Universal Robots PolyScope program: g_2.urp

Program g_2 (installation=string_planes directory=/programs createdIn=5.17.3 lastSavedIn=5.17.3 robotSerialNumber=20245501435)
Calibrated DH parameters: a=[0.000154, -0.137004, -0.385524, -0.00002, 0.000092, 0]; d=[0.162441, 211.794786, -230.585024, 18.923638, 0.099786, 0.09951]; alpha=[1.569493, -0.001902, 0.003874, 1.570111, -1.570167, 0]; deltaTheta=[0, -1.242934, 1.056292, 0.186646, 0.000002, 0.000001]
InitVariablesNode
Robot Program (runOnlyOnce=false)
  MoveL speed 250 mm/s, acceleration 1200 mm/s^2 (useActiveTCP=true) feature=Plane_3
    Waypoint Waypoint_1: TCP in base x=347.51 y=672.22 z=96.15 mm, rx=-1.6525 ry=-1.6511 rz=0.6428 rad; joints [-132.145, -24.912, 67.944, -99.663, -48.733, -144.753] deg; TCP offset x=28.21 y=-96.107 z=-99.69 mm, rx=0 ry=0 rz=0 rad; feature pose in base x=319.452 y=675.799 z=94.591 mm, rx=2.7302 ry=-0.0495 rz=1.4252 rad
    Waypoint Waypoint_2 (Relative): relativeFromPosition TCP in base x=347.532 y=672.21 z=96.159 mm, rx=-1.6525 ry=-1.6511 rz=0.6428 rad; joints [-132.146, -24.912, 67.943, -99.662, -48.733, -144.753] deg; TCP in base x=328.782 y=410.687 z=69.436 mm, rx=-1.5068 ry=-1.7187 rz=0.8745 rad; joints [-148.419, -39.387, 107.724, -104.601, -66.349, -167.764] deg
